// Mitsubishi GX Works2 project: BookEX6_30 Logical   PLC: Q13UDV

// global labels: Global
VAR_GLOBAL
  bVar0 AT M5000 : BOOL;
  abArray0 AT M5010 : ARRAY [0..49] OF BOOL;
  sStr0 AT D5000 : STRING[199];
  sStr1 AT D5100 : STRING[199];
  sStr2 AT D5200 : STRING[199];
  sStr3 AT D5300 : STRING[199];
  sStr4 AT D5400 : STRING[199];
  sStr5 AT D5500 : STRING[199];
  sStr6 AT D5600 : STRING[199];
  sStr7 AT D5700 : STRING[199];
  sStr8 AT D5800 : STRING[199];
  sStr9 AT D5900 : STRING[199];
  iVar0 AT D4500 : INT;
  iVar1 AT D4501 : INT;
  iVar2 AT D4502 : INT;
  iVar3 AT D4503 : INT;
  iVar4 AT D4504 : INT;
  iVar5 AT D4505 : INT;
  iVar6 AT D4506 : INT;
  iVar7 AT D4507 : INT;
  iVar8 AT D4508 : INT;
  iVar9 AT D4509 : INT;
  dVar0 AT D4510 : DINT;
  dVar1 AT D4512 : DINT;
  dVar2 AT D4514 : DINT;
  dVar3 AT D4516 : DINT;
  dVar4 AT D4518 : DINT;
  dVar5 AT D4520 : DINT;
  dVar6 AT D4522 : DINT;
  dVar7 AT D4524 : DINT;
  dVar8 AT D4526 : DINT;
  dVar9 AT D4528 : DINT;
  wVar0 AT D4530 : WORD;
  wVar1 AT D4531 : WORD;
  wVar2 AT D4532 : WORD;
  wVar3 AT D4533 : WORD;
  wVar4 AT D4534 : WORD;
  wVar5 AT D4535 : WORD;
  wVar6 AT D4536 : WORD;
  wVar7 AT D4537 : WORD;
  wVar8 AT D4538 : WORD;
  wVar9 AT D4539 : WORD;
  dwVar0 AT D4540 : DWORD;
  dwVar1 AT D4542 : DWORD;
  dwVar2 AT D4544 : DWORD;
  dwVar3 AT D4546 : DWORD;
  dwVar4 AT D4548 : DWORD;
  dwVar5 AT D4550 : DWORD;
  dwVar6 AT D4552 : DWORD;
  dwVar7 AT D4554 : DWORD;
  dwVar8 AT D4556 : DWORD;
  dwVar9 AT D4558 : DWORD;
  fsVar0 AT D4560 : REAL;
  fsVar1 AT D4562 : REAL;
  fsVar2 AT D4564 : REAL;
  fsVar3 AT D4566 : REAL;
  fsVar4 AT D4568 : REAL;
  fsVar5 AT D4570 : REAL;
  fsVar6 AT D4572 : REAL;
  fsVar7 AT D4574 : REAL;
  fsVar8 AT D4576 : REAL;
  fsVar9 AT D4578 : REAL;
  fdVar0 AT D4580 : LREAL;
  tTime0 AT D4620 : TIME;
  tTime1 AT D4622 : TIME;
  tTime2 AT D4624 : TIME;
  tTime3 AT D4626 : TIME;
  tTime4 AT D4628 : TIME;
  tTime5 AT D4630 : TIME;
  tTime6 AT D4632 : TIME;
  tTime7 AT D4634 : TIME;
  tTime8 AT D4636 : TIME;
  tTime9 AT D4638 : TIME;
  tTime10 AT D4640 : TIME;
  bVar1 AT M5001 : BOOL;
  bVar2 AT M5002 : BOOL;
  bVar3 AT M5003 : BOOL;
  bVar4 AT M5004 : BOOL;
  bVar5 AT M5005 : BOOL;
  bVar6 AT M5006 : BOOL;
  bVar7 AT M5007 : BOOL;
  bVar8 AT M5008 : BOOL;
  bVar9 AT M5009 : BOOL;
  abArray1 AT M5060 : ARRAY [0..49] OF BOOL;
  abArray2 AT M5110 : ARRAY [0..49] OF BOOL;
  abArray3 AT M5160 : ARRAY [0..49] OF BOOL;
  abArray4 AT M5210 : ARRAY [0..49] OF BOOL;
  abArray5 AT M5260 : ARRAY [0..49] OF BOOL;
  abArray6 AT M5310 : ARRAY [0..49] OF BOOL;
  abArray7 AT M5360 : ARRAY [0..49] OF BOOL;
  abArray8 AT M5410 : ARRAY [0..49] OF BOOL;
  abArray9 AT M5460 : ARRAY [0..49] OF BOOL;
  fdVar1 AT D4584 : LREAL;
  fdVar2 AT D4588 : LREAL;
  fdVar3 AT D4592 : LREAL;
  fdVar4 AT D4596 : LREAL;
  fdVar5 AT D4600 : LREAL;
  fdVar6 AT D4604 : LREAL;
  fdVar7 AT D4608 : LREAL;
  fdVar8 AT D4612 : LREAL;
  fdVar9 AT D4616 : LREAL;
  afsPen0 AT D2000 : ARRAY [0..499] OF REAL;
  afsPen1 AT D3000 : ARRAY [0..499] OF REAL;
END_VAR
// user libraries (not included): HMI

FUNCTION OffBitWORD
VAR_INPUT
  w_IN : WORD;
  i_POS : INT;
END_VAR
VAR
  w_DATA : WORD;
END_VAR
;
w_DATA := H0001;
SFL(TRUE, i_POS, w_DATA);
OffBitWORD := w_IN AND NOT w_DATA;
END_FUNCTION

FUNCTION OnBitWORD
VAR_INPUT
  w_IN : WORD;
  i_POS : INT;
END_VAR
VAR
  w_DATA : WORD;
END_VAR
;
w_DATA := H0001;
SFL(TRUE, i_POS, w_DATA);
OnBitWORD := w_IN OR w_DATA;
END_FUNCTION

FUNCTION ToggBitWORD
VAR_INPUT
  w_IN : WORD;
  i_POS : INT;
END_VAR
VAR
  w_DATA : WORD;
END_VAR
;
w_DATA := H0001;
SFL(TRUE, i_POS, w_DATA);
ToggBitWORD := w_IN XOR w_DATA;
END_FUNCTION

PROGRAM ExBIT_WORD
(* structured ladder/FBD written out as ST: instructions are called as NAME(EN, inputs, outputs); _pN, _eN, _tN stand for wires *)
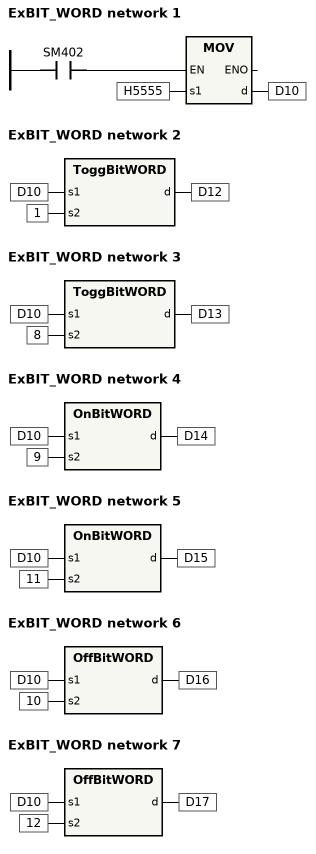
(* network 1 *)
MOV(SM402, H5555, D10);
(* network 2 *)
D12 := ToggBitWORD(D10, 1);
(* network 3 *)
D13 := ToggBitWORD(D10, 8);
(* network 4 *)
D14 := OnBitWORD(D10, 9);
(* network 5 *)
D15 := OnBitWORD(D10, 11);
(* network 6 *)
D16 := OffBitWORD(D10, 10);
(* network 7 *)
D17 := OffBitWORD(D10, 12);
END_PROGRAM

PROGRAM ExBKAND
VAR
  Mov4WORD_1 : Mov4WORD;
  Mov4WORD_2 : Mov4WORD;
  Mov4WORD_3 : Mov4WORD;
  Mov4WORD_4 : Mov4WORD;
END_VAR
(* structured ladder/FBD written out as ST: instructions are called as NAME(EN, inputs, outputs); _pN, _eN, _tN stand for wires *)
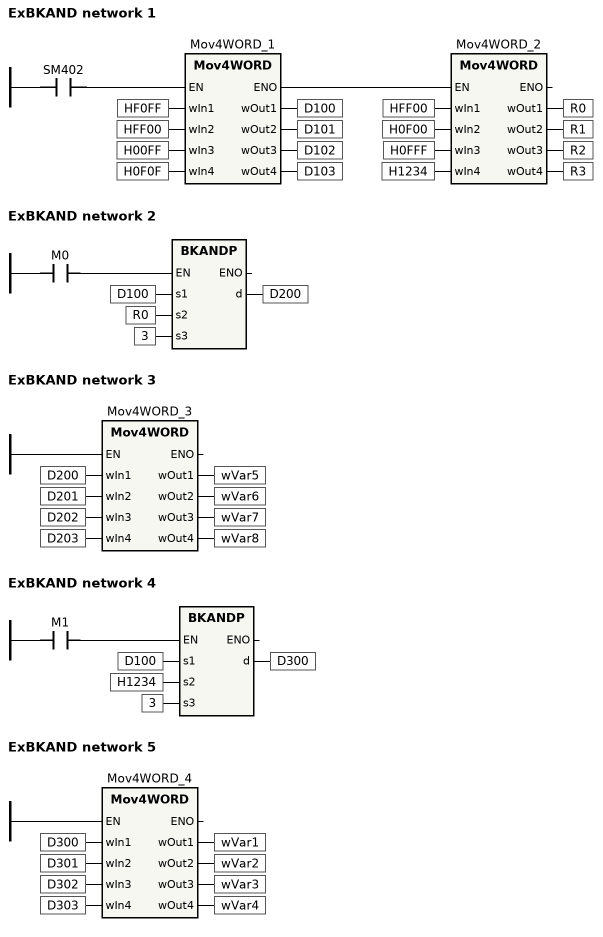
(* network 1 *)
Mov4WORD_1(EN := SM402, wIn1 := HF0FF, wIn2 := HFF00, wIn3 := H00FF, wIn4 := H0F0F, wOut1 => D100, wOut2 => D101, wOut3 => D102, wOut4 => D103);
Mov4WORD_2(EN := Mov4WORD_1.ENO, wIn1 := HFF00, wIn2 := H0F00, wIn3 := H0FFF, wIn4 := H1234, wOut1 => R0, wOut2 => R1, wOut3 => R2, wOut4 => R3);
(* network 2 *)
BKANDP(M0, D100, R0, 3, D200);
(* network 3 *)
Mov4WORD_3(EN := TRUE, wIn1 := D200, wIn2 := D201, wIn3 := D202, wIn4 := D203, wOut1 => wVar5, wOut2 => wVar6, wOut3 => wVar7, wOut4 => wVar8);
(* network 4 *)
BKANDP(M1, D100, H1234, 3, D300);
(* network 5 *)
Mov4WORD_4(EN := TRUE, wIn1 := D300, wIn2 := D301, wIn3 := D302, wIn4 := D303, wOut1 => wVar1, wOut2 => wVar2, wOut3 => wVar3, wOut4 => wVar4);
END_PROGRAM

PROGRAM ExBKOR
VAR
  Mov4WORD_1 : Mov4WORD;
  Mov4WORD_2 : Mov4WORD;
  Mov4WORD_3 : Mov4WORD;
  Mov4WORD_4 : Mov4WORD;
END_VAR
(* structured ladder/FBD written out as ST: instructions are called as NAME(EN, inputs, outputs); _pN, _eN, _tN stand for wires *)
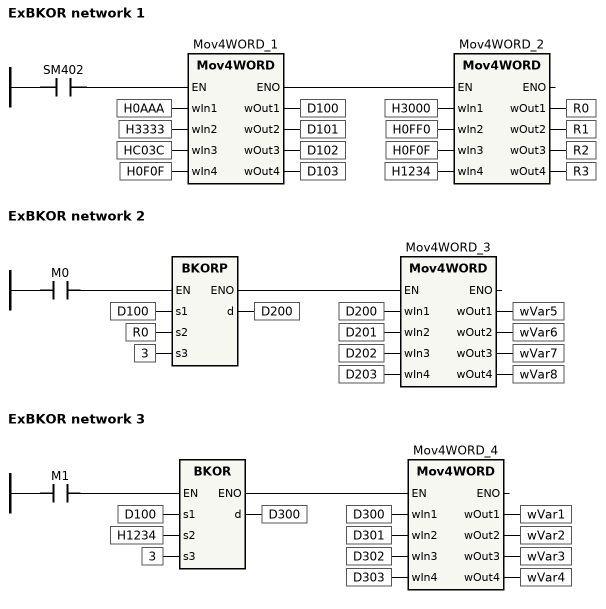
(* network 1 *)
Mov4WORD_1(EN := SM402, wIn1 := H0AAA, wIn2 := H3333, wIn3 := HC03C, wIn4 := H0F0F, wOut1 => D100, wOut2 => D101, wOut3 => D102, wOut4 => D103);
Mov4WORD_2(EN := Mov4WORD_1.ENO, wIn1 := H3000, wIn2 := H0FF0, wIn3 := H0F0F, wIn4 := H1234, wOut1 => R0, wOut2 => R1, wOut3 => R2, wOut4 => R3);
(* network 2 *)
_e1 := BKORP(M0, D100, R0, 3, D200);
Mov4WORD_3(EN := _e1, wIn1 := D200, wIn2 := D201, wIn3 := D202, wIn4 := D203, wOut1 => wVar5, wOut2 => wVar6, wOut3 => wVar7, wOut4 => wVar8);
(* network 3 *)
_e1 := BKOR(M1, D100, H1234, 3, D300);
Mov4WORD_4(EN := _e1, wIn1 := D300, wIn2 := D301, wIn3 := D302, wIn4 := D303, wOut1 => wVar1, wOut2 => wVar2, wOut3 => wVar3, wOut4 => wVar4);
END_PROGRAM

PROGRAM ExBKXNR
VAR
  Mov4WORD_1 : Mov4WORD;
  Mov4WORD_2 : Mov4WORD;
  Mov4WORD_3 : Mov4WORD;
  Mov4WORD_4 : Mov4WORD;
END_VAR
(* structured ladder/FBD written out as ST: instructions are called as NAME(EN, inputs, outputs); _pN, _eN, _tN stand for wires *)
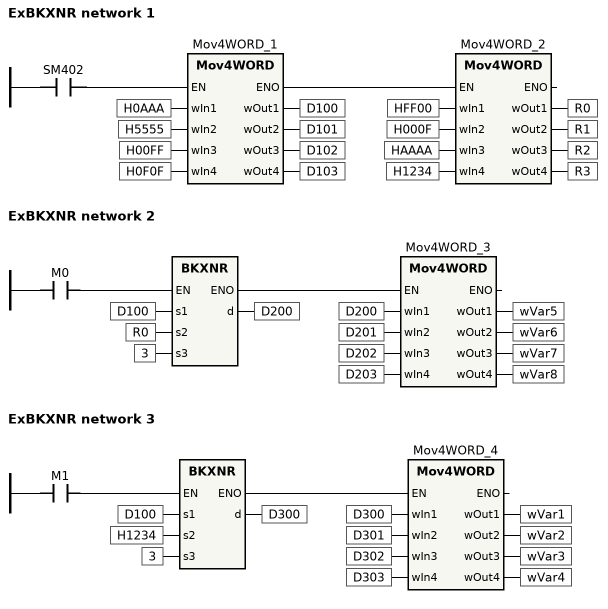
(* network 1 *)
Mov4WORD_1(EN := SM402, wIn1 := H0AAA, wIn2 := H5555, wIn3 := H00FF, wIn4 := H0F0F, wOut1 => D100, wOut2 => D101, wOut3 => D102, wOut4 => D103);
Mov4WORD_2(EN := Mov4WORD_1.ENO, wIn1 := HFF00, wIn2 := H000F, wIn3 := HAAAA, wIn4 := H1234, wOut1 => R0, wOut2 => R1, wOut3 => R2, wOut4 => R3);
(* network 2 *)
_e1 := BKXNR(M0, D100, R0, 3, D200);
Mov4WORD_3(EN := _e1, wIn1 := D200, wIn2 := D201, wIn3 := D202, wIn4 := D203, wOut1 => wVar5, wOut2 => wVar6, wOut3 => wVar7, wOut4 => wVar8);
(* network 3 *)
_e1 := BKXNR(M1, D100, H1234, 3, D300);
Mov4WORD_4(EN := _e1, wIn1 := D300, wIn2 := D301, wIn3 := D302, wIn4 := D303, wOut1 => wVar1, wOut2 => wVar2, wOut3 => wVar3, wOut4 => wVar4);
END_PROGRAM

PROGRAM ExBKXOR
VAR
  Mov4WORD_1 : Mov4WORD;
  Mov4WORD_2 : Mov4WORD;
  Mov4WORD_3 : Mov4WORD;
  Mov4WORD_4 : Mov4WORD;
END_VAR
(* structured ladder/FBD written out as ST: instructions are called as NAME(EN, inputs, outputs); _pN, _eN, _tN stand for wires *)
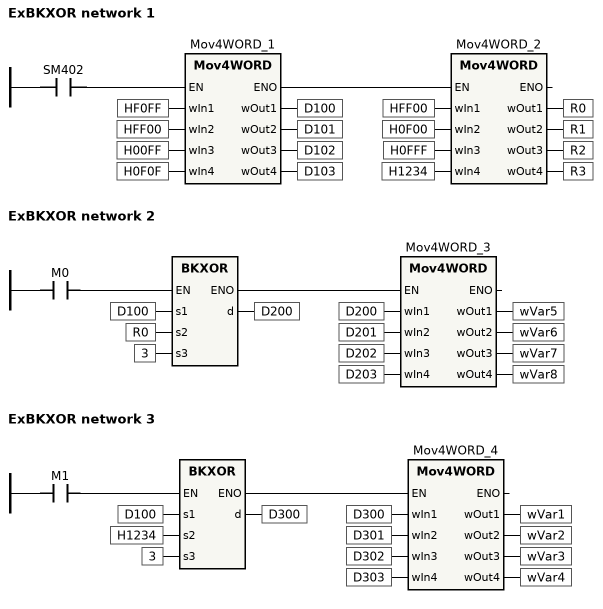
(* network 1 *)
Mov4WORD_1(EN := SM402, wIn1 := HF0FF, wIn2 := HFF00, wIn3 := H00FF, wIn4 := H0F0F, wOut1 => D100, wOut2 => D101, wOut3 => D102, wOut4 => D103);
Mov4WORD_2(EN := Mov4WORD_1.ENO, wIn1 := HFF00, wIn2 := H0F00, wIn3 := H0FFF, wIn4 := H1234, wOut1 => R0, wOut2 => R1, wOut3 => R2, wOut4 => R3);
(* network 2 *)
_e1 := BKXOR(M0, D100, R0, 3, D200);
Mov4WORD_3(EN := _e1, wIn1 := D200, wIn2 := D201, wIn3 := D202, wIn4 := D203, wOut1 => wVar5, wOut2 => wVar6, wOut3 => wVar7, wOut4 => wVar8);
(* network 3 *)
_e1 := BKXOR(M1, D100, H1234, 3, D300);
Mov4WORD_4(EN := _e1, wIn1 := D300, wIn2 := D301, wIn3 := D302, wIn4 := D303, wOut1 => wVar1, wOut2 => wVar2, wOut3 => wVar3, wOut4 => wVar4);
END_PROGRAM

PROGRAM ExWAND
(* structured ladder/FBD written out as ST: instructions are called as NAME(EN, inputs, outputs); _pN, _eN, _tN stand for wires *)
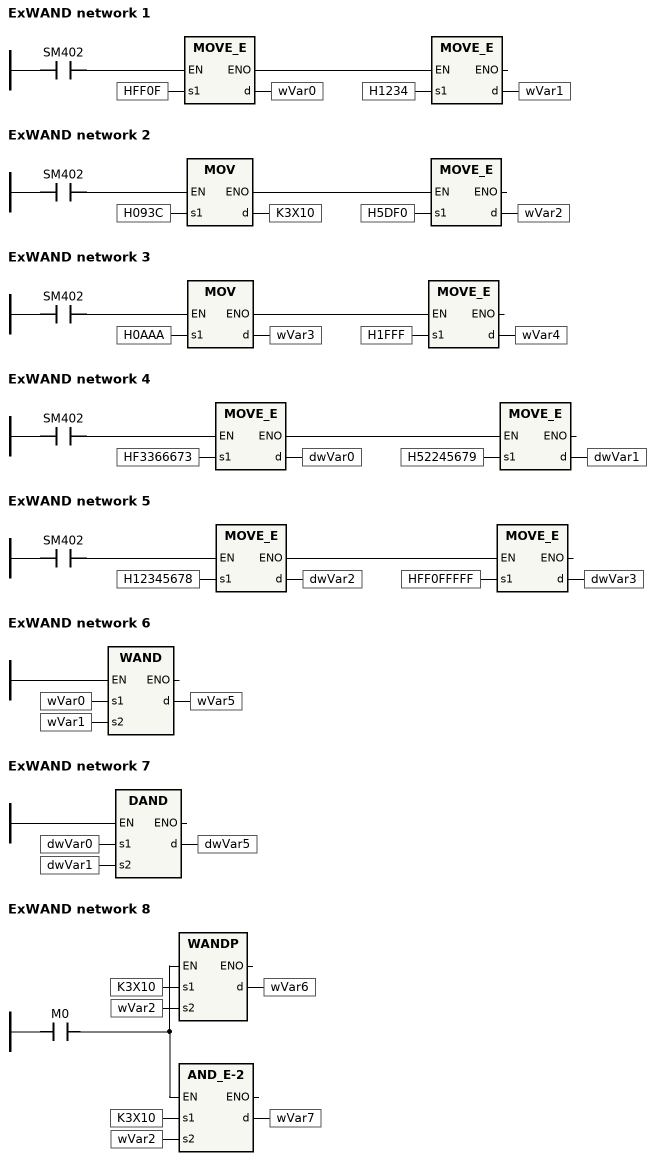
(* network 1 *)
_e1 := MOVE_E(SM402, HFF0F, wVar0);
MOVE_E(_e1, H1234, wVar1);
(* network 2 *)
_e1 := MOV(SM402, H093C, K3X10);
MOVE_E(_e1, H5DF0, wVar2);
(* network 3 *)
_e1 := MOV(SM402, H0AAA, wVar3);
MOVE_E(_e1, H1FFF, wVar4);
(* network 4 *)
_e1 := MOVE_E(SM402, HF3366673, dwVar0);
MOVE_E(_e1, H52245679, dwVar1);
(* network 5 *)
_e1 := MOVE_E(SM402, H12345678, dwVar2);
MOVE_E(_e1, HFF0FFFFF, dwVar3);
(* network 6 *)
WAND(TRUE, wVar0, wVar1, wVar5);
(* network 7 *)
DAND(TRUE, dwVar0, dwVar1, dwVar5);
(* network 8 *)
WANDP(M0, K3X10, wVar2, wVar6);
AND_E(M0, K3X10, wVar2, wVar7);
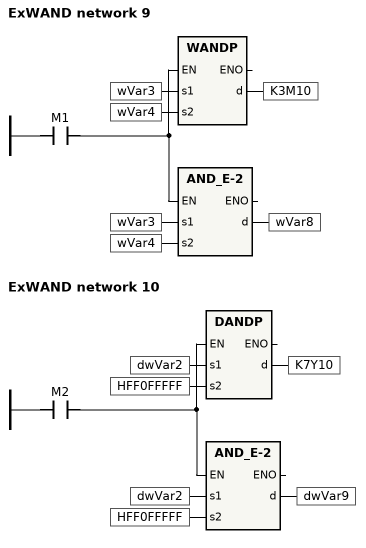
(* network 9 *)
WANDP(M1, wVar3, wVar4, K3M10);
AND_E(M1, wVar3, wVar4, wVar8);
(* network 10 *)
DANDP(M2, dwVar2, HFF0FFFFF, K7Y10);
AND_E(M2, dwVar2, HFF0FFFFF, dwVar9);
END_PROGRAM

PROGRAM ExWOR
(* structured ladder/FBD written out as ST: instructions are called as NAME(EN, inputs, outputs); _pN, _eN, _tN stand for wires *)
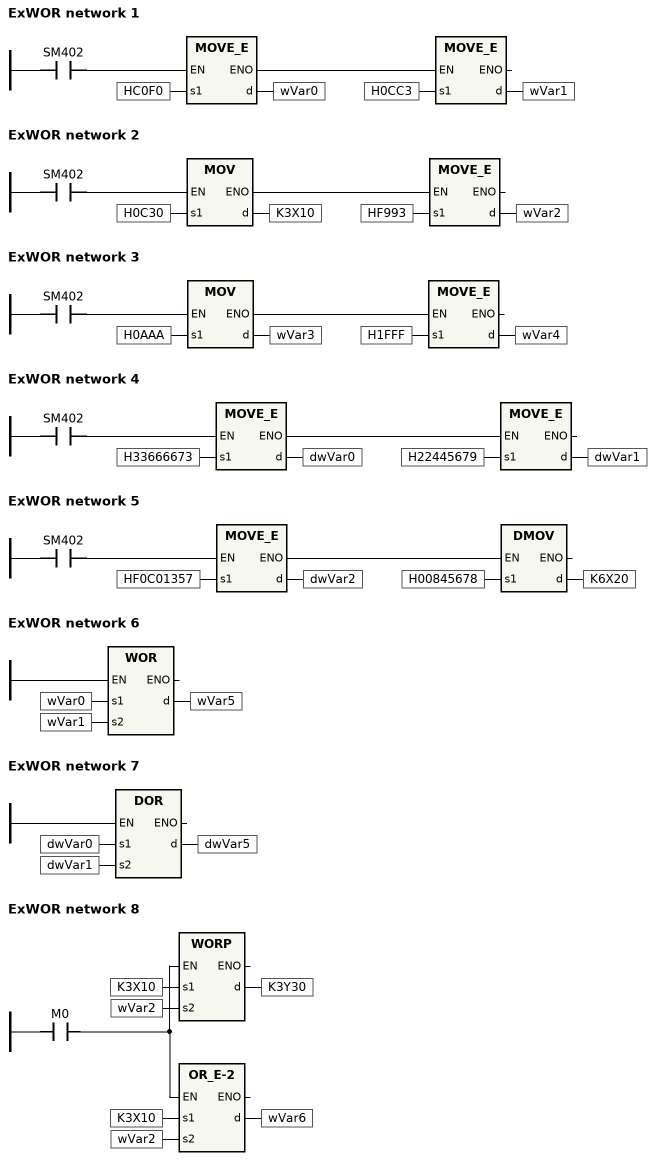
(* network 1 *)
_e1 := MOVE_E(SM402, HC0F0, wVar0);
MOVE_E(_e1, H0CC3, wVar1);
(* network 2 *)
_e1 := MOV(SM402, H0C30, K3X10);
MOVE_E(_e1, HF993, wVar2);
(* network 3 *)
_e1 := MOV(SM402, H0AAA, wVar3);
MOVE_E(_e1, H1FFF, wVar4);
(* network 4 *)
_e1 := MOVE_E(SM402, H33666673, dwVar0);
MOVE_E(_e1, H22445679, dwVar1);
(* network 5 *)
_e1 := MOVE_E(SM402, HF0C01357, dwVar2);
DMOV(_e1, H00845678, K6X20);
(* network 6 *)
WOR(TRUE, wVar0, wVar1, wVar5);
(* network 7 *)
DOR(TRUE, dwVar0, dwVar1, dwVar5);
(* network 8 *)
WORP(M0, K3X10, wVar2, K3Y30);
OR_E(M0, K3X10, wVar2, wVar6);
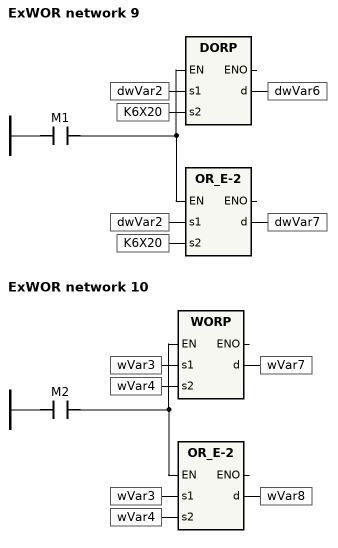
(* network 9 *)
DORP(M1, dwVar2, K6X20, dwVar6);
OR_E(M1, dwVar2, K6X20, dwVar7);
(* network 10 *)
WORP(M2, wVar3, wVar4, wVar7);
OR_E(M2, wVar3, wVar4, wVar8);
END_PROGRAM

PROGRAM ExWXNR
(* structured ladder/FBD written out as ST: instructions are called as NAME(EN, inputs, outputs); _pN, _eN, _tN stand for wires *)
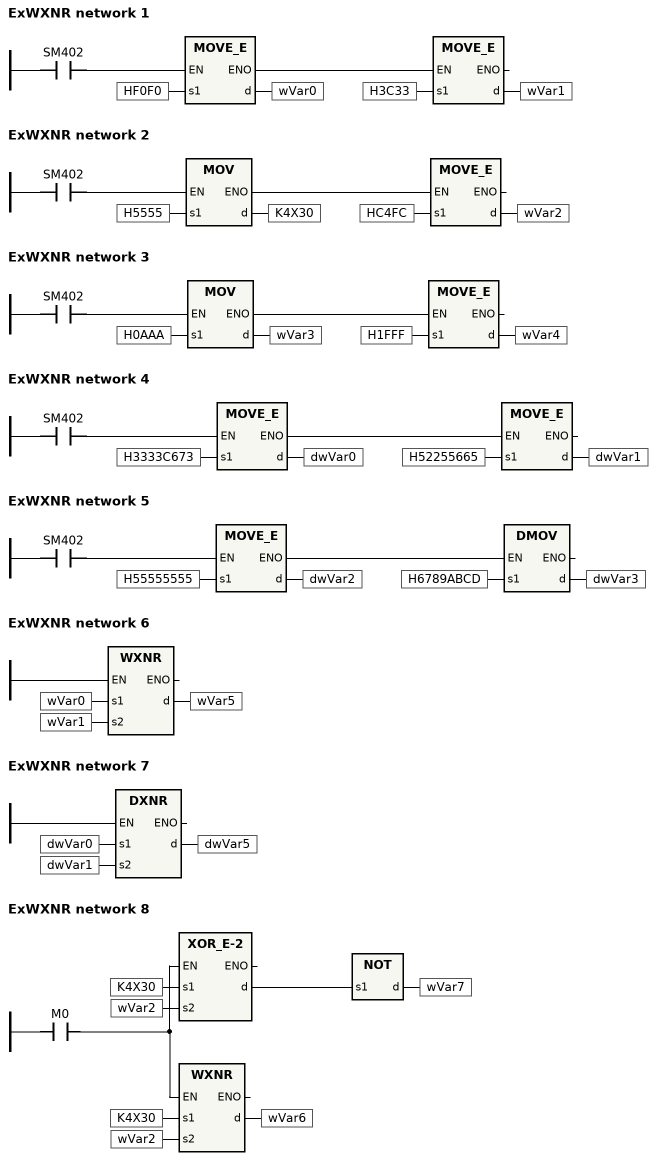
(* network 1 *)
_e1 := MOVE_E(SM402, HF0F0, wVar0);
MOVE_E(_e1, H3C33, wVar1);
(* network 2 *)
_e1 := MOV(SM402, H5555, K4X30);
MOVE_E(_e1, HC4FC, wVar2);
(* network 3 *)
_e1 := MOV(SM402, H0AAA, wVar3);
MOVE_E(_e1, H1FFF, wVar4);
(* network 4 *)
_e1 := MOVE_E(SM402, H3333C673, dwVar0);
MOVE_E(_e1, H52255665, dwVar1);
(* network 5 *)
_e1 := MOVE_E(SM402, H55555555, dwVar2);
DMOV(_e1, H6789ABCD, dwVar3);
(* network 6 *)
WXNR(TRUE, wVar0, wVar1, wVar5);
(* network 7 *)
DXNR(TRUE, dwVar0, dwVar1, dwVar5);
(* network 8 *)
WXNR(M0, K4X30, wVar2, wVar6);
XOR_E(M0, K4X30, wVar2, _t1);
wVar7 := NOT(_t1);
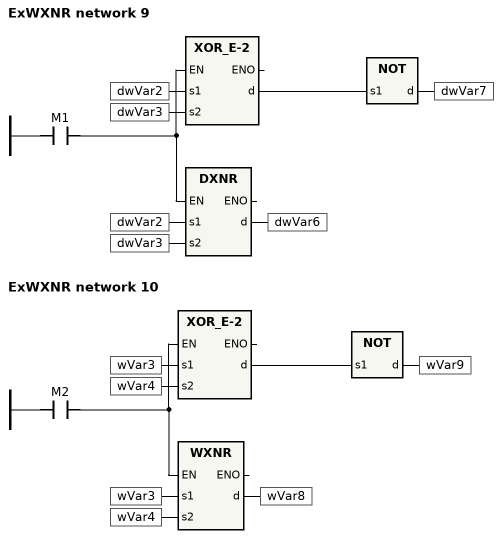
(* network 9 *)
DXNR(M1, dwVar2, dwVar3, dwVar6);
XOR_E(M1, dwVar2, dwVar3, _t1);
dwVar7 := NOT(_t1);
(* network 10 *)
WXNR(M2, wVar3, wVar4, wVar8);
XOR_E(M2, wVar3, wVar4, _t1);
wVar9 := NOT(_t1);
END_PROGRAM

PROGRAM ExWXOR
(* structured ladder/FBD written out as ST: instructions are called as NAME(EN, inputs, outputs); _pN, _eN, _tN stand for wires *)
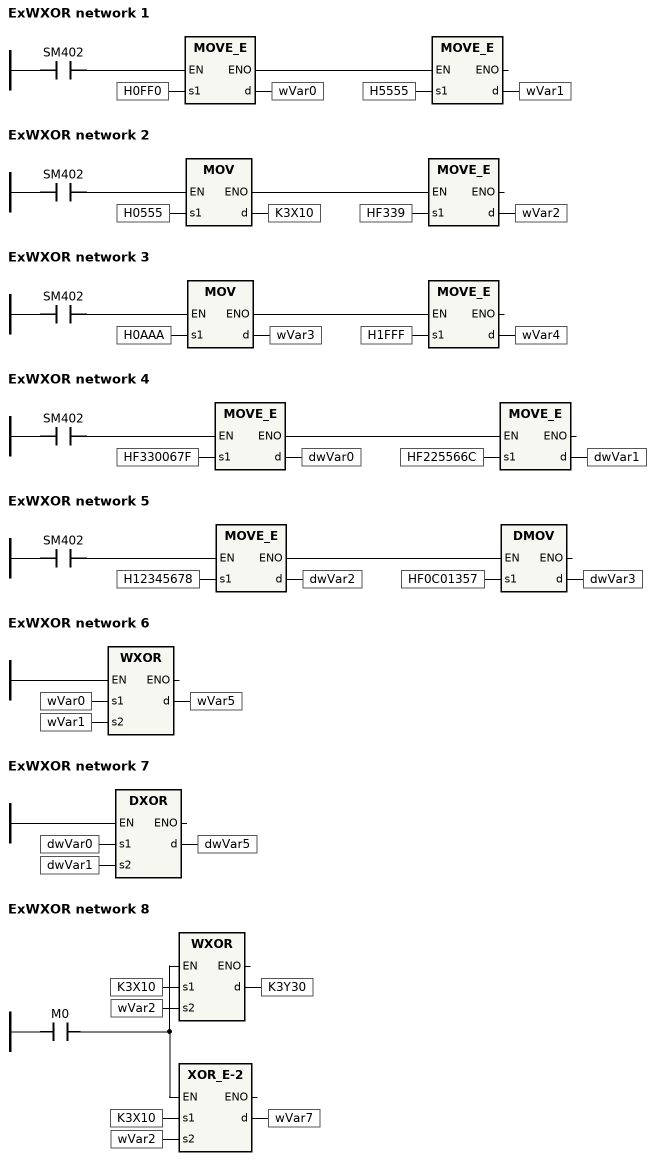
(* network 1 *)
_e1 := MOVE_E(SM402, H0FF0, wVar0);
MOVE_E(_e1, H5555, wVar1);
(* network 2 *)
_e1 := MOV(SM402, H0555, K3X10);
MOVE_E(_e1, HF339, wVar2);
(* network 3 *)
_e1 := MOV(SM402, H0AAA, wVar3);
MOVE_E(_e1, H1FFF, wVar4);
(* network 4 *)
_e1 := MOVE_E(SM402, HF330067F, dwVar0);
MOVE_E(_e1, HF225566C, dwVar1);
(* network 5 *)
_e1 := MOVE_E(SM402, H12345678, dwVar2);
DMOV(_e1, HF0C01357, dwVar3);
(* network 6 *)
WXOR(TRUE, wVar0, wVar1, wVar5);
(* network 7 *)
DXOR(TRUE, dwVar0, dwVar1, dwVar5);
(* network 8 *)
WXOR(M0, K3X10, wVar2, K3Y30);
XOR_E(M0, K3X10, wVar2, wVar7);
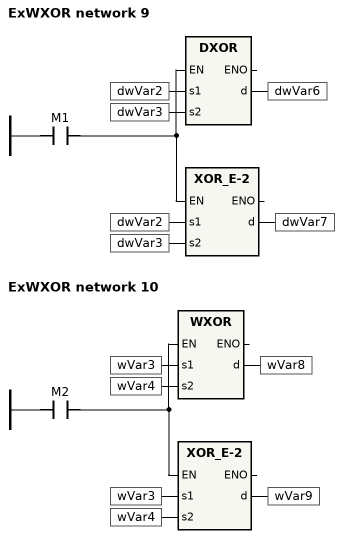
(* network 9 *)
DXOR(M1, dwVar2, dwVar3, dwVar6);
XOR_E(M1, dwVar2, dwVar3, dwVar7);
(* network 10 *)
WXOR(M2, wVar3, wVar4, wVar8);
XOR_E(M2, wVar3, wVar4, wVar9);
END_PROGRAM
